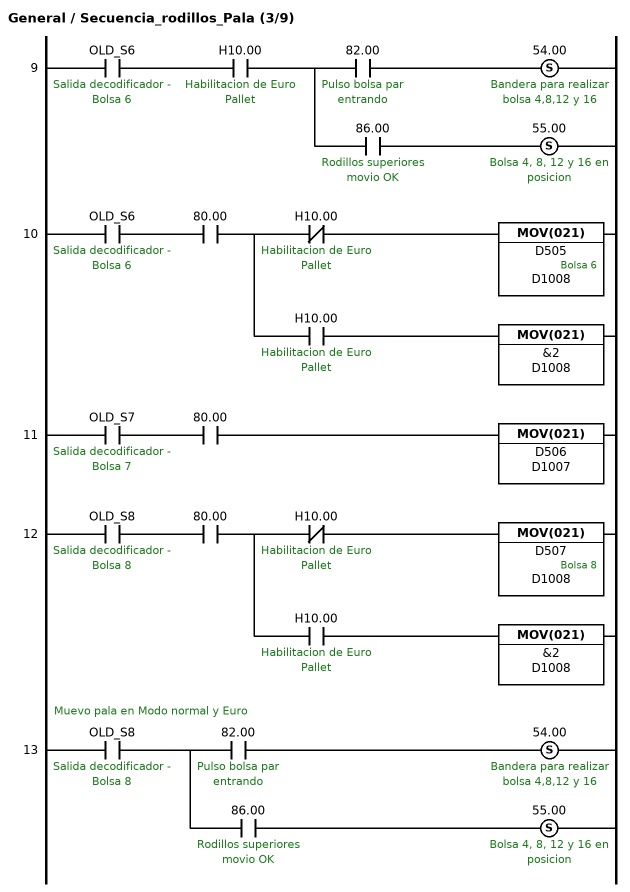
; [picture p48: General / Secuencia_rodillos_Pala, rungs 9-13]
; rung 9
LD OLD_S6  ; Salida decodificador - Bolsa 6
AND H10.00  ; Habilitacion de Euro Pallet
OUT TR0
AND 82.00  ; Pulso bolsa par entrando
SET 54.00  ; Bandera para realizar bolsa 4,8,12 y 16
LD TR0
AND 86.00  ; Rodillos superiores movio OK
SET 55.00  ; Bolsa 4, 8, 12 y 16 en posicion
; rung 10
LD OLD_S6  ; Salida decodificador - Bolsa 6
AND 80.00
OUT TR0
ANDNOT H10.00  ; Habilitacion de Euro Pallet
MOV(021) D505 D1008  ; Bolsa 6
LD TR0
AND H10.00  ; Habilitacion de Euro Pallet
MOV(021) &2 D1008
; rung 11
LD OLD_S7  ; Salida decodificador - Bolsa 7
AND 80.00
MOV(021) D506 D1007
; rung 12
LD OLD_S8  ; Salida decodificador - Bolsa 8
AND 80.00
OUT TR0
ANDNOT H10.00  ; Habilitacion de Euro Pallet
MOV(021) D507 D1008  ; Bolsa 8  // Original valor &8
LD TR0
AND H10.00  ; Habilitacion de Euro Pallet
MOV(021) &2 D1008  // Original valor &8
; rung 13: Muevo pala en Modo normal y Euro
LD OLD_S8  ; Salida decodificador - Bolsa 8
OUT TR0
AND 82.00  ; Pulso bolsa par entrando
SET 54.00  ; Bandera para realizar bolsa 4,8,12 y 16
LD TR0
AND 86.00  ; Rodillos superiores movio OK
SET 55.00  ; Bolsa 4, 8, 12 y 16 en posicion

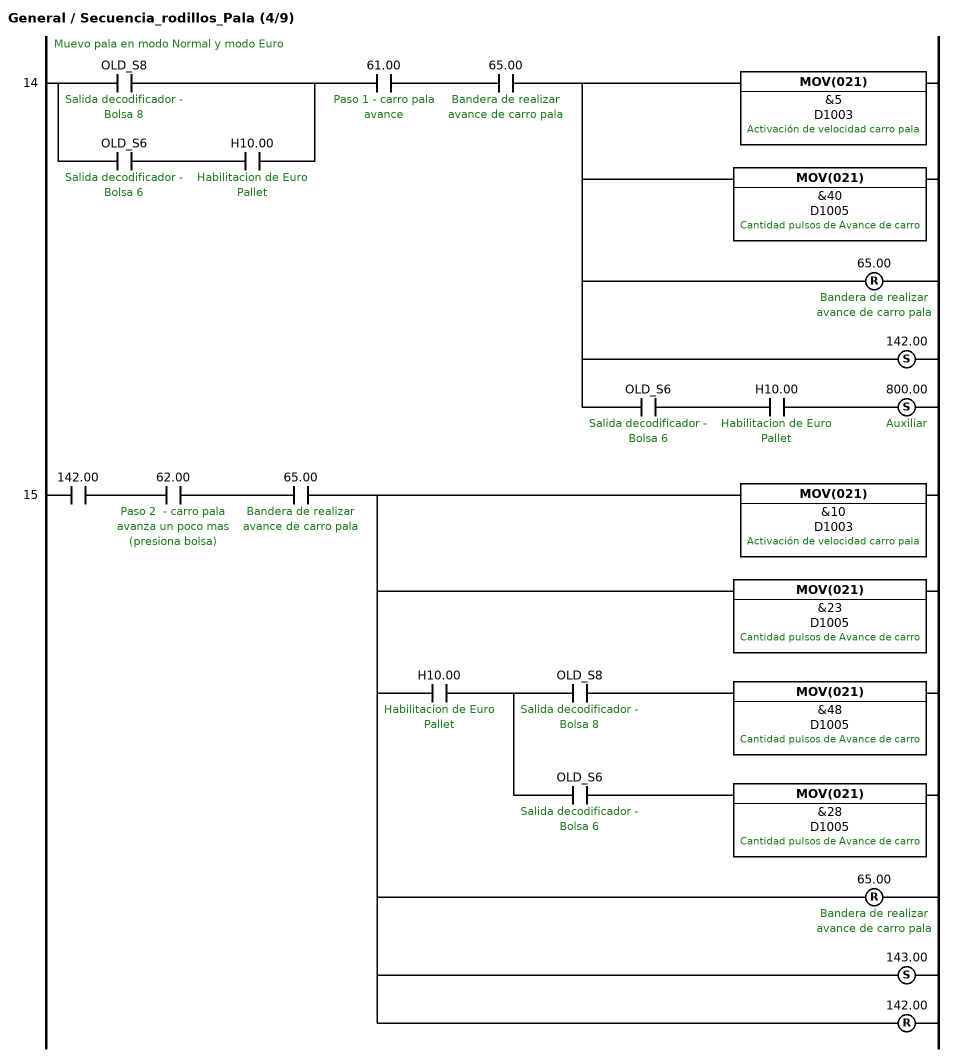
; rung 14: Muevo pala en modo Normal y modo Euro
LD OLD_S8  ; Salida decodificador - Bolsa 8
LD OLD_S6  ; Salida decodificador - Bolsa 6
AND H10.00  ; Habilitacion de Euro Pallet
ORLD
AND 61.00  ; Paso 1 - carro pala avance
AND 65.00  ; Bandera de realizar avance de carro pala
MOV(021) &5 D1003  ; Activación de velocidad carro pala
MOV(021) &40 D1005  ; Cantidad pulsos de Avance de carro
RSET 65.00  ; Bandera de realizar avance de carro pala
SET 142.00
AND OLD_S6  ; Salida decodificador - Bolsa 6
AND H10.00  ; Habilitacion de Euro Pallet
SET 800.00  ; Auxiliar
; rung 15
LD 142.00
AND 62.00  ; Paso 2  - carro pala avanza un poco mas (presiona bolsa)
AND 65.00  ; Bandera de realizar avance de carro pala
OUT TR0
MOV(021) &10 D1003  ; Activación de velocidad carro pala
MOV(021) &23 D1005  ; Cantidad pulsos de Avance de carro
AND H10.00  ; Habilitacion de Euro Pallet
OUT TR1
AND OLD_S8  ; Salida decodificador - Bolsa 8
MOV(021) &48 D1005  ; Cantidad pulsos de Avance de carro
LD TR1
AND OLD_S6  ; Salida decodificador - Bolsa 6
MOV(021) &28 D1005  ; Cantidad pulsos de Avance de carro
LD TR0
RSET 65.00  ; Bandera de realizar avance de carro pala
SET 143.00
RSET 142.00

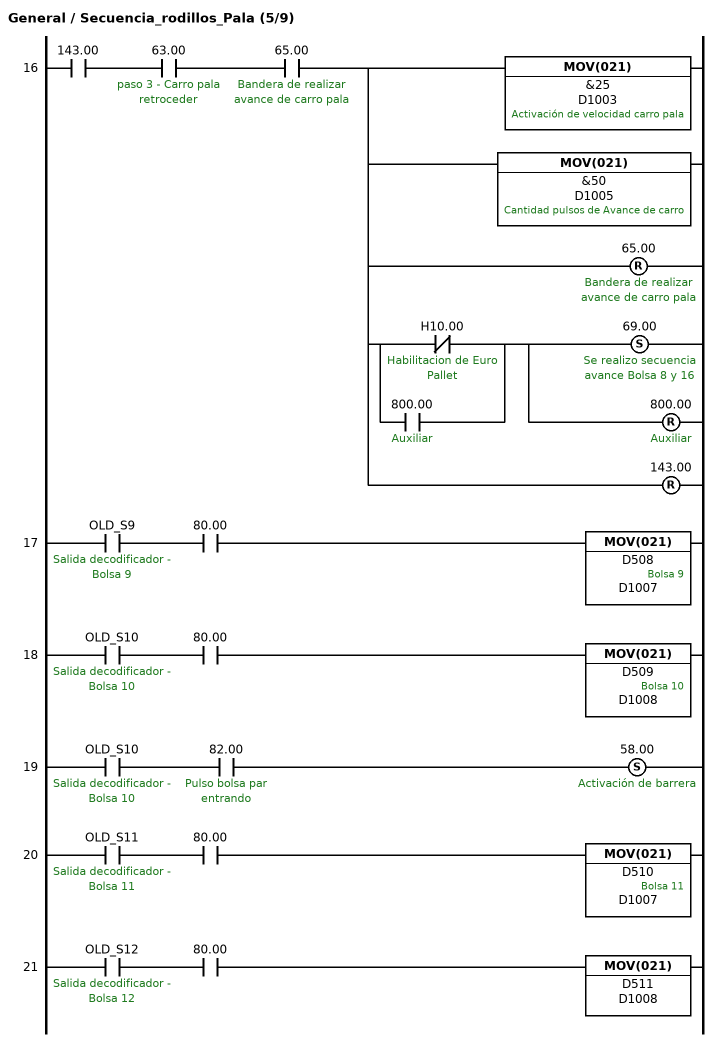
; rung 16
LD 143.00
AND 63.00  ; paso 3 - Carro pala retroceder
AND 65.00  ; Bandera de realizar avance de carro pala
OUT TR0
MOV(021) &25 D1003  ; Activación de velocidad carro pala
MOV(021) &50 D1005  ; Cantidad pulsos de Avance de carro
RSET 65.00  ; Bandera de realizar avance de carro pala
LDNOT H10.00  ; Habilitacion de Euro Pallet
OR 800.00  ; Auxiliar
ANDLD
SET 69.00  ; Se realizo secuencia avance Bolsa 8 y 16
RSET 800.00  ; Auxiliar
LD TR0
RSET 143.00
; rung 17
LD OLD_S9  ; Salida decodificador - Bolsa 9
AND 80.00
MOV(021) D508 D1007  ; Bolsa 9
; rung 18
LD OLD_S10  ; Salida decodificador - Bolsa 10
AND 80.00
MOV(021) D509 D1008  ; Bolsa 10
; rung 19
LD OLD_S10  ; Salida decodificador - Bolsa 10
AND 82.00  ; Pulso bolsa par entrando
SET 58.00  ; Activación de barrera
; rung 20
LD OLD_S11  ; Salida decodificador - Bolsa 11
AND 80.00
MOV(021) D510 D1007  ; Bolsa 11
; rung 21
LD OLD_S12  ; Salida decodificador - Bolsa 12
AND 80.00
MOV(021) D511 D1008

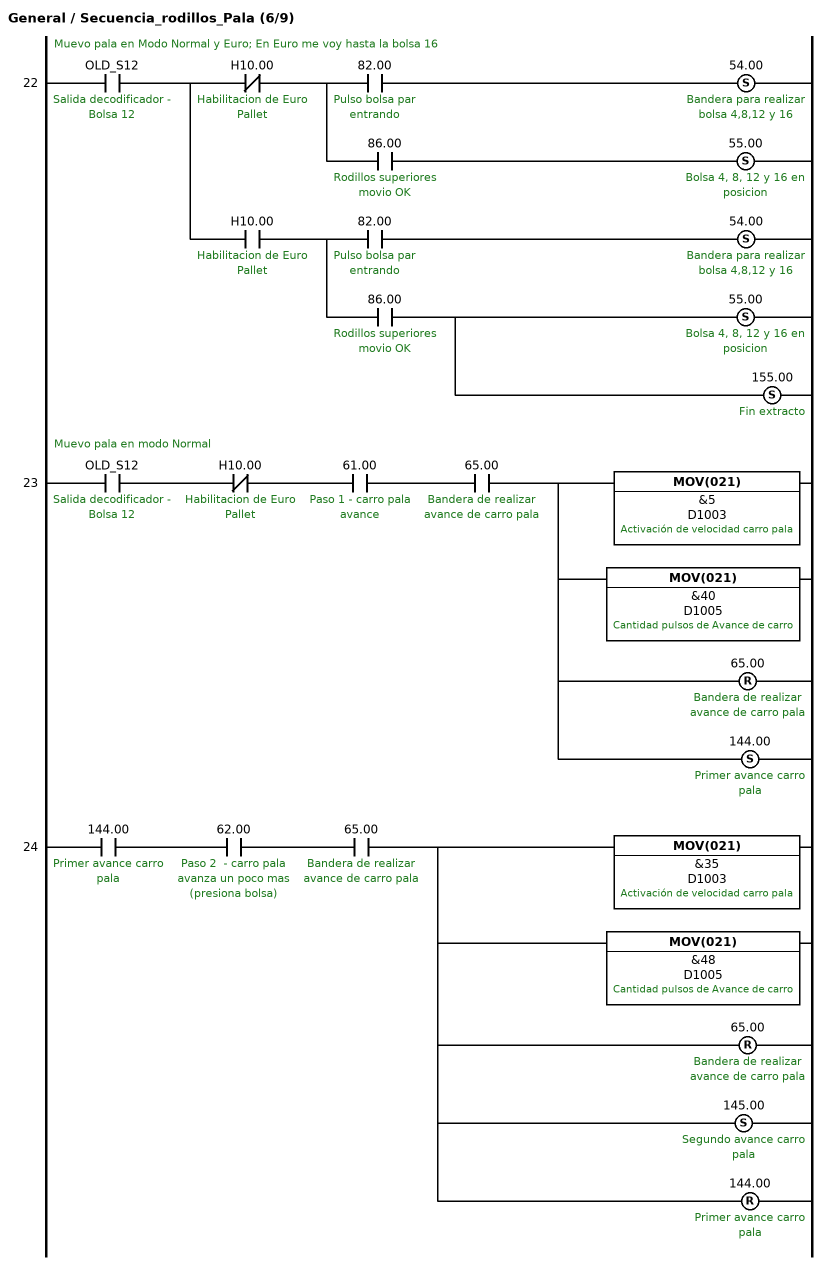
; rung 22: Muevo pala en Modo Normal y Euro; En Euro me voy hasta la bolsa 16
LD OLD_S12  ; Salida decodificador - Bolsa 12
OUT TR0
ANDNOT H10.00  ; Habilitacion de Euro Pallet
OUT TR1
AND 82.00  ; Pulso bolsa par entrando
SET 54.00  ; Bandera para realizar bolsa 4,8,12 y 16
LD TR1
AND 86.00  ; Rodillos superiores movio OK
SET 55.00  ; Bolsa 4, 8, 12 y 16 en posicion
LD TR0
AND H10.00  ; Habilitacion de Euro Pallet
OUT TR0
AND 82.00  ; Pulso bolsa par entrando
SET 54.00  ; Bandera para realizar bolsa 4,8,12 y 16
LD TR0
AND 86.00  ; Rodillos superiores movio OK
SET 55.00  ; Bolsa 4, 8, 12 y 16 en posicion
SET 155.00  ; Fin extracto
; rung 23: Muevo pala en modo Normal
LD OLD_S12  ; Salida decodificador - Bolsa 12
ANDNOT H10.00  ; Habilitacion de Euro Pallet
AND 61.00  ; Paso 1 - carro pala avance
AND 65.00  ; Bandera de realizar avance de carro pala
MOV(021) &5 D1003  ; Activación de velocidad carro pala
MOV(021) &40 D1005  ; Cantidad pulsos de Avance de carro
RSET 65.00  ; Bandera de realizar avance de carro pala
SET 144.00  ; Primer avance carro pala
; rung 24
LD 144.00  ; Primer avance carro pala
AND 62.00  ; Paso 2  - carro pala avanza un poco mas (presiona bolsa)
AND 65.00  ; Bandera de realizar avance de carro pala
MOV(021) &35 D1003  ; Activación de velocidad carro pala
MOV(021) &48 D1005  ; Cantidad pulsos de Avance de carro
RSET 65.00  ; Bandera de realizar avance de carro pala
SET 145.00  ; Segundo avance carro pala
RSET 144.00  ; Primer avance carro pala

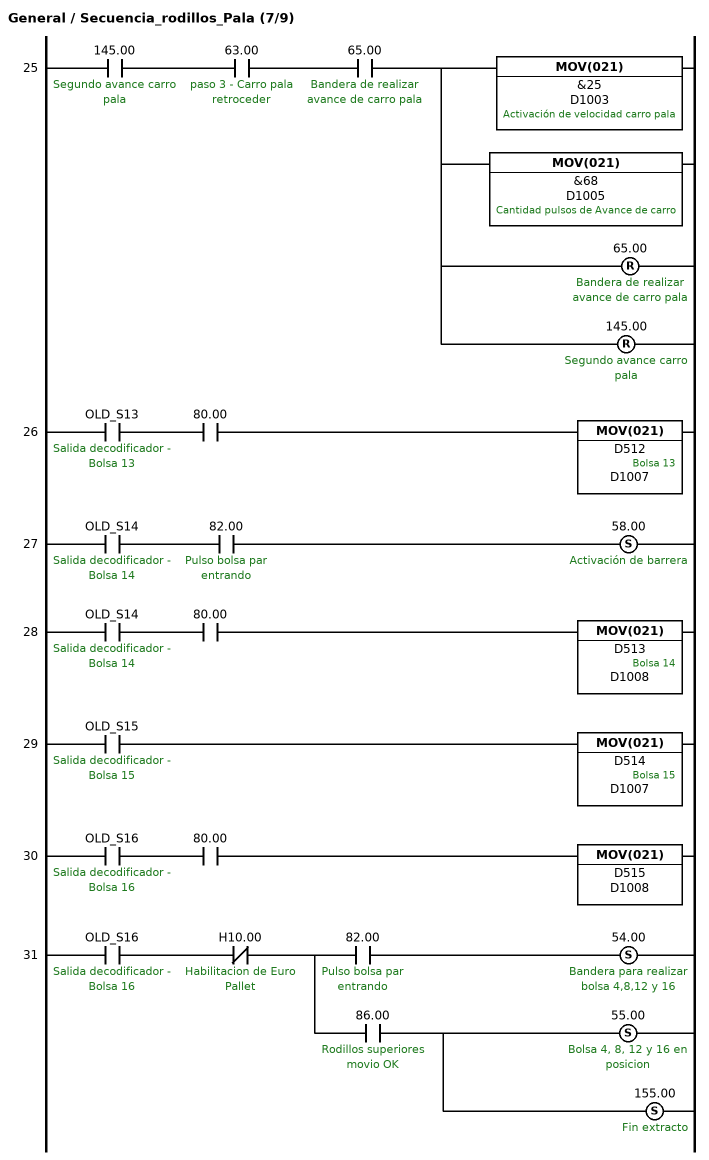
; rung 25
LD 145.00  ; Segundo avance carro pala
AND 63.00  ; paso 3 - Carro pala retroceder
AND 65.00  ; Bandera de realizar avance de carro pala
MOV(021) &25 D1003  ; Activación de velocidad carro pala
MOV(021) &68 D1005  ; Cantidad pulsos de Avance de carro
RSET 65.00  ; Bandera de realizar avance de carro pala
RSET 145.00  ; Segundo avance carro pala
; rung 26
LD OLD_S13  ; Salida decodificador - Bolsa 13
AND 80.00
MOV(021) D512 D1007  ; Bolsa 13
; rung 27
LD OLD_S14  ; Salida decodificador - Bolsa 14
AND 82.00  ; Pulso bolsa par entrando
SET 58.00  ; Activación de barrera
; rung 28
LD OLD_S14  ; Salida decodificador - Bolsa 14
AND 80.00
MOV(021) D513 D1008  ; Bolsa 14
; rung 29
LD OLD_S15  ; Salida decodificador - Bolsa 15
MOV(021) D514 D1007  ; Bolsa 15
; rung 30
LD OLD_S16  ; Salida decodificador - Bolsa 16
AND 80.00
MOV(021) D515 D1008  // Original valor &6
; rung 31
LD OLD_S16  ; Salida decodificador - Bolsa 16
ANDNOT H10.00  ; Habilitacion de Euro Pallet
OUT TR0
AND 82.00  ; Pulso bolsa par entrando
SET 54.00  ; Bandera para realizar bolsa 4,8,12 y 16
LD TR0
AND 86.00  ; Rodillos superiores movio OK
SET 55.00  ; Bolsa 4, 8, 12 y 16 en posicion
SET 155.00  ; Fin extracto

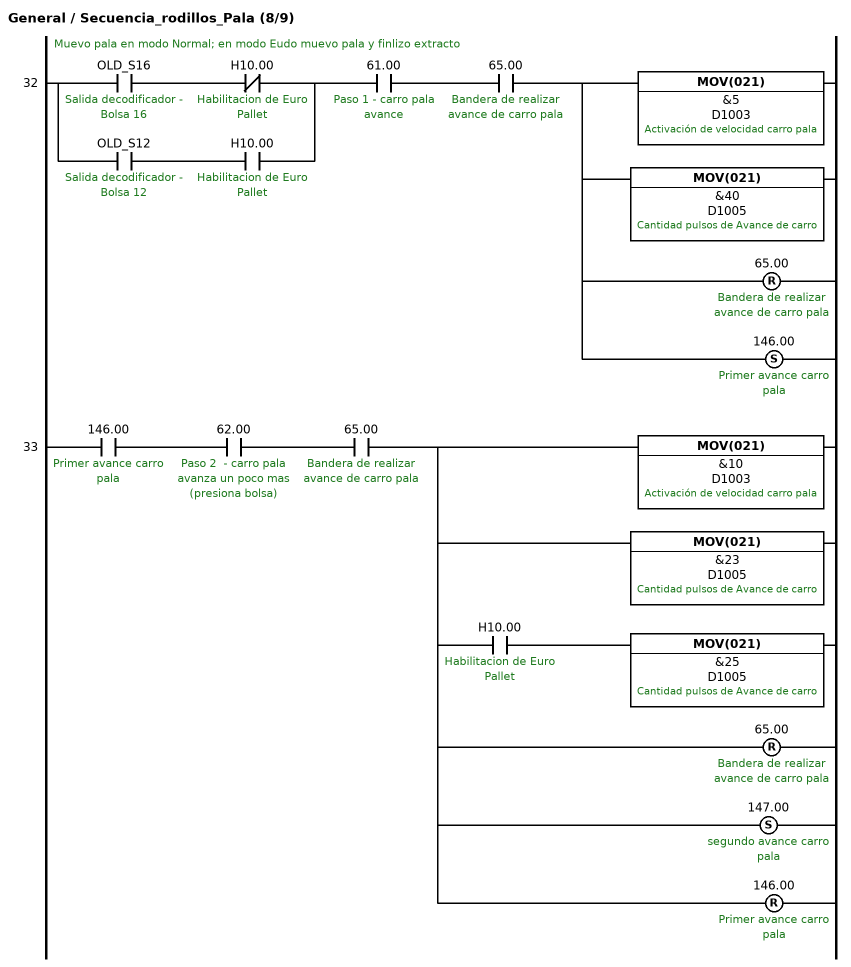
; rung 32: Muevo pala en modo Normal; en modo Eudo muevo pala y finlizo extracto
LD OLD_S16  ; Salida decodificador - Bolsa 16
ANDNOT H10.00  ; Habilitacion de Euro Pallet
LD OLD_S12  ; Salida decodificador - Bolsa 12
AND H10.00  ; Habilitacion de Euro Pallet
ORLD
AND 61.00  ; Paso 1 - carro pala avance
AND 65.00  ; Bandera de realizar avance de carro pala
MOV(021) &5 D1003  ; Activación de velocidad carro pala
MOV(021) &40 D1005  ; Cantidad pulsos de Avance de carro
RSET 65.00  ; Bandera de realizar avance de carro pala
SET 146.00  ; Primer avance carro pala
; rung 33
LD 146.00  ; Primer avance carro pala
AND 62.00  ; Paso 2  - carro pala avanza un poco mas (presiona bolsa)
AND 65.00  ; Bandera de realizar avance de carro pala
OUT TR0
MOV(021) &10 D1003  ; Activación de velocidad carro pala
MOV(021) &23 D1005  ; Cantidad pulsos de Avance de carro
AND H10.00  ; Habilitacion de Euro Pallet
MOV(021) &25 D1005  ; Cantidad pulsos de Avance de carro
LD TR0
RSET 65.00  ; Bandera de realizar avance de carro pala
SET 147.00  ; segundo avance carro pala
RSET 146.00  ; Primer avance carro pala

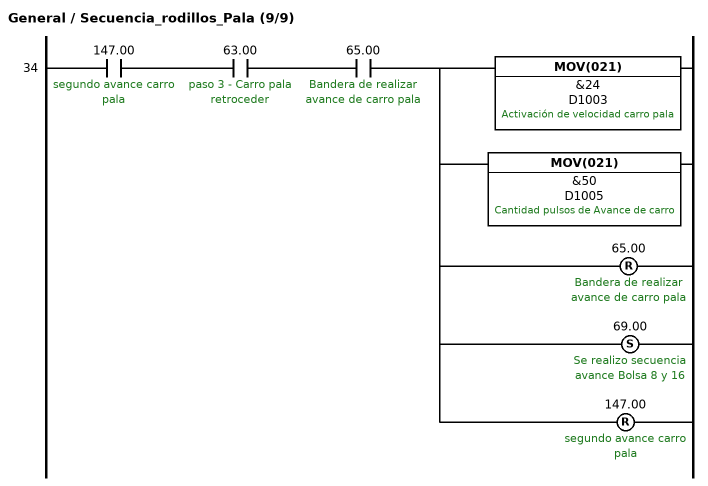
; rung 34
LD 147.00  ; segundo avance carro pala
AND 63.00  ; paso 3 - Carro pala retroceder
AND 65.00  ; Bandera de realizar avance de carro pala
MOV(021) &24 D1003  ; Activación de velocidad carro pala
MOV(021) &50 D1005  ; Cantidad pulsos de Avance de carro
RSET 65.00  ; Bandera de realizar avance de carro pala
SET 69.00  ; Se realizo secuencia avance Bolsa 8 y 16
RSET 147.00  ; segundo avance carro pala

### Section _Fin_Salto

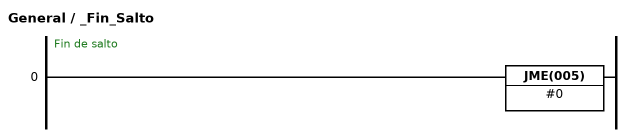
; rung 0: Fin de salto
JME(005) #0

### Section Habilitaciones_MAN_AUT

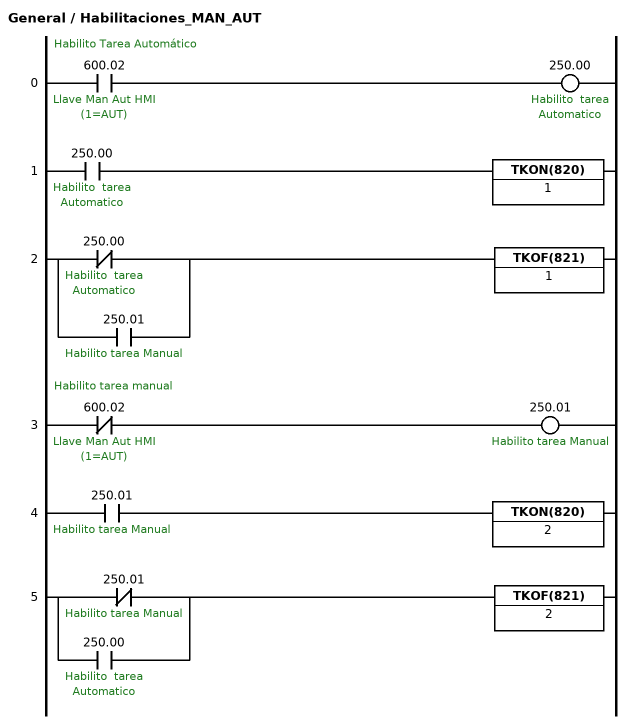
; rung 0: Habilito Tarea Automático
LD 600.02  ; Llave Man Aut HMI (1=AUT)
OUT 250.00  ; Habilito  tarea Automatico
; rung 1
LD 250.00  ; Habilito  tarea Automatico
TKON(820) 1
; rung 2
LDNOT 250.00  ; Habilito  tarea Automatico
OR 250.01  ; Habilito tarea Manual
TKOF(821) 1
; rung 3: Habilito tarea manual
LDNOT 600.02  ; Llave Man Aut HMI (1=AUT)
OUT 250.01  ; Habilito tarea Manual
; rung 4
LD 250.01  ; Habilito tarea Manual
TKON(820) 2
; rung 5
LDNOT 250.01  ; Habilito tarea Manual
OR 250.00  ; Habilito  tarea Automatico
TKOF(821) 2

### Section Seleccion_pallet

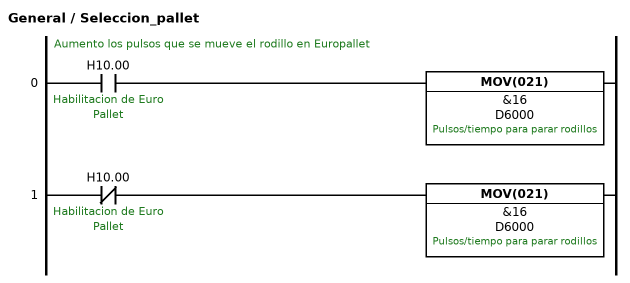
; rung 0: Aumento los pulsos que se mueve el rodillo en Europallet
LD H10.00  ; Habilitacion de Euro Pallet
MOV(021) &16 D6000  ; Pulsos/tiempo para parar rodillos
; rung 1
LDNOT H10.00  ; Habilitacion de Euro Pallet
MOV(021) &16 D6000  ; Pulsos/tiempo para parar rodillos

### Section Señales_enfundora

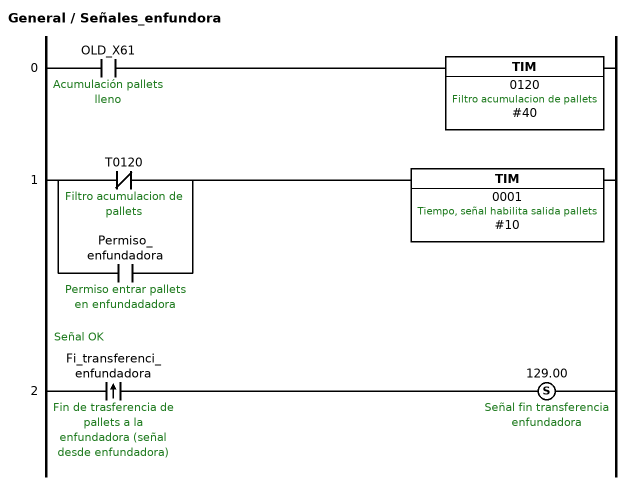
; rung 0
LD OLD_X61  ; Acumulación pallets lleno
TIM 0120 #40  ; Filtro acumulacion de pallets
; rung 1
LDNOT T0120  ; Filtro acumulacion de pallets
OR Permiso_enfundadora  ; Permiso entrar pallets en enfundadadora
TIM 0001 #10  ; Tiempo, señal habilita salida pallets
; rung 2: Señal OK
@LD Fi_transferenci_enfundadora  ; Fin de trasferencia de pallets a la enfundadora (señal desde enfundadora)
SET 129.00  ; Señal fin transferencia enfundadora

### Section Alarmas

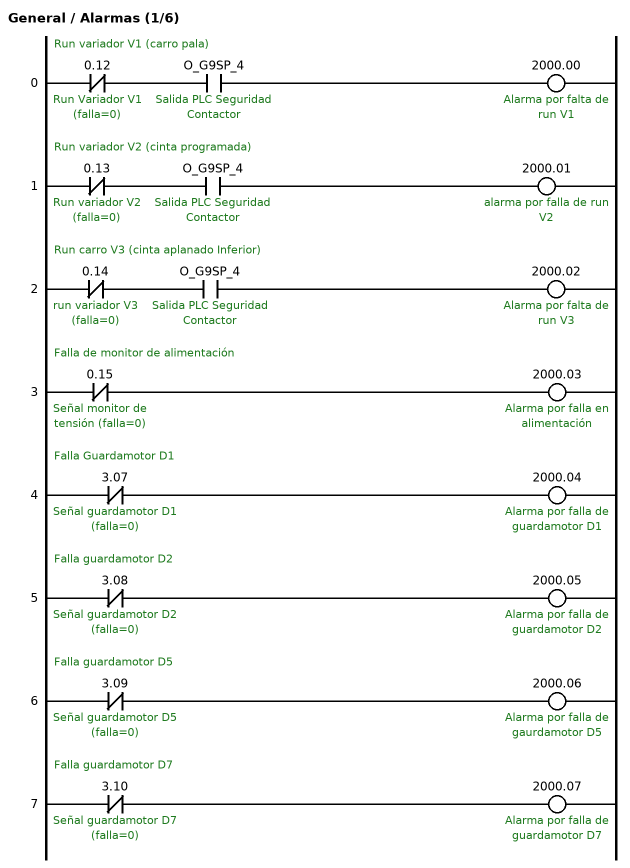
; rung 0: Run variador V1 (carro pala)
LDNOT 0.12  ; Run Variador V1 (falla=0)
AND O_G9SP_4  ; Salida PLC Seguridad Contactor
OUT 2000.00  ; Alarma por falta de run V1
; rung 1: Run variador V2 (cinta programada)
LDNOT 0.13  ; Run variador V2 (falla=0)
AND O_G9SP_4  ; Salida PLC Seguridad Contactor
OUT 2000.01  ; alarma por falla de run V2
; rung 2: Run carro V3 (cinta aplanado Inferior)
LDNOT 0.14  ; run variador V3 (falla=0)
AND O_G9SP_4  ; Salida PLC Seguridad Contactor
OUT 2000.02  ; Alarma por falta de run V3
; rung 3: Falla de monitor de alimentación
LDNOT 0.15  ; Señal monitor de tensión (falla=0)
OUT 2000.03  ; Alarma por falla en alimentación
; rung 4: Falla Guardamotor D1
LDNOT 3.07  ; Señal guardamotor D1 (falla=0)
OUT 2000.04  ; Alarma por falla de guardamotor D1
; rung 5: Falla guardamotor D2
LDNOT 3.08  ; Señal guardamotor D2 (falla=0)
OUT 2000.05  ; Alarma por falla de guardamotor D2
; rung 6: Falla guardamotor D5
LDNOT 3.09  ; Señal guardamotor D5 (falla=0)
OUT 2000.06  ; Alarma por falla de gaurdamotor D5
; rung 7: Falla guardamotor D7
LDNOT 3.10  ; Señal guardamotor D7 (falla=0)
OUT 2000.07  ; Alarma por falla de guardamotor D7

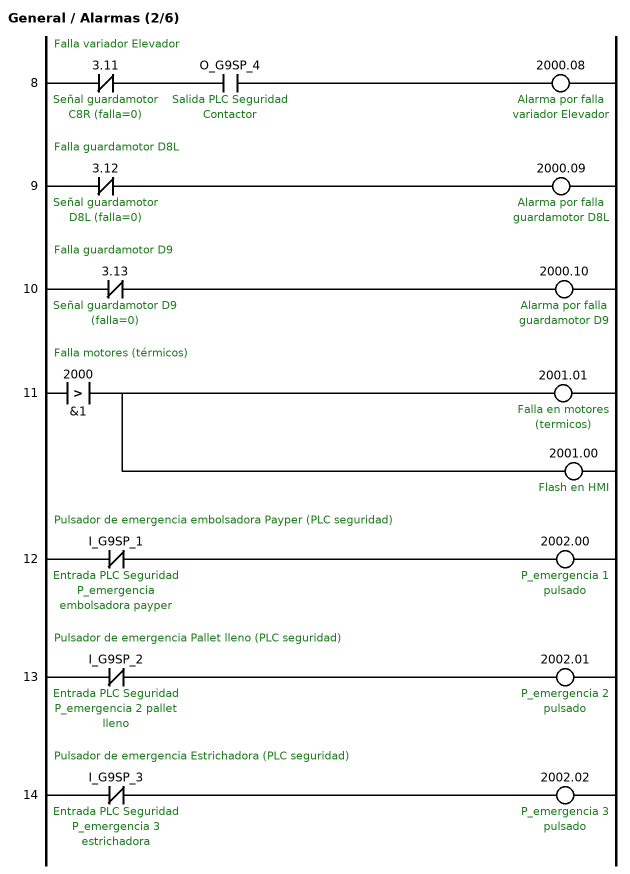
; rung 8: Falla variador Elevador
LDNOT 3.11  ; Señal guardamotor C8R (falla=0)
AND O_G9SP_4  ; Salida PLC Seguridad Contactor
OUT 2000.08  ; Alarma por falla variador Elevador
; rung 9: Falla guardamotor D8L
LDNOT 3.12  ; Señal guardamotor D8L (falla=0)
OUT 2000.09  ; Alarma por falla guardamotor D8L
; rung 10: Falla guardamotor D9
LDNOT 3.13  ; Señal guardamotor D9 (falla=0)
OUT 2000.10  ; Alarma por falla guardamotor D9
; rung 11: Falla motores (térmicos)
LD>(320) 2000 &1
OUT 2001.01  ; Falla en motores (termicos)
OUT 2001.00  ; Flash en HMI
; rung 12: Pulsador de emergencia embolsadora Payper (PLC seguridad)
LDNOT I_G9SP_1  ; Entrada PLC Seguridad P_emergencia embolsadora payper
OUT 2002.00  ; P_emergencia 1 pulsado
; rung 13: Pulsador de emergencia Pallet lleno (PLC seguridad)
LDNOT I_G9SP_2  ; Entrada PLC Seguridad P_emergencia 2 pallet lleno
OUT 2002.01  ; P_emergencia 2 pulsado
; rung 14: Pulsador de emergencia Estrichadora (PLC seguridad)
LDNOT I_G9SP_3  ; Entrada PLC Seguridad P_emergencia 3 estrichadora
OUT 2002.02  ; P_emergencia 3 pulsado

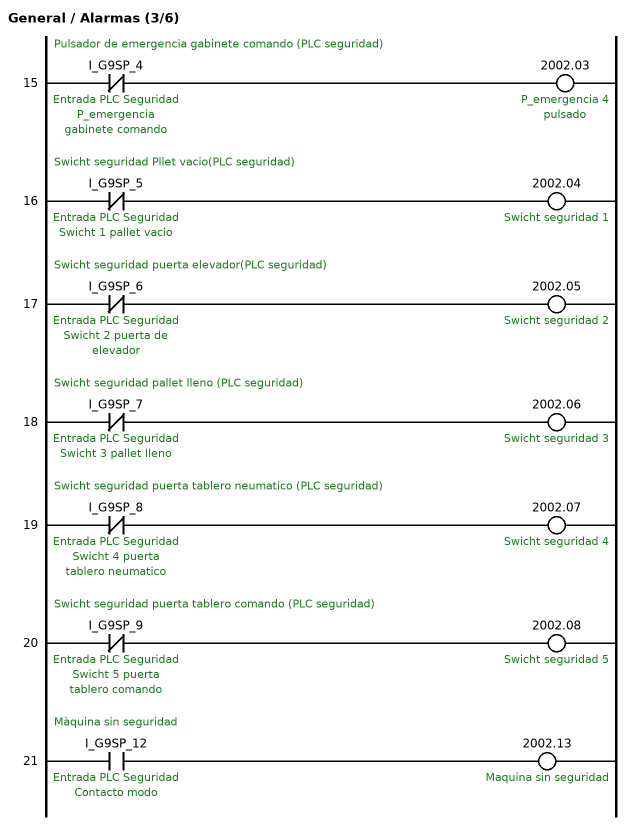
; rung 15: Pulsador de emergencia gabinete comando (PLC seguridad)
LDNOT I_G9SP_4  ; Entrada PLC Seguridad P_emergencia gabinete comando
OUT 2002.03  ; P_emergencia 4 pulsado
; rung 16: Swicht seguridad Pllet vacio(PLC seguridad)
LDNOT I_G9SP_5  ; Entrada PLC Seguridad Swicht 1 pallet vacio
OUT 2002.04  ; Swicht seguridad 1
; rung 17: Swicht seguridad puerta elevador(PLC seguridad)
LDNOT I_G9SP_6  ; Entrada PLC Seguridad Swicht 2 puerta de elevador
OUT 2002.05  ; Swicht seguridad 2
; rung 18: Swicht seguridad pallet lleno (PLC seguridad)
LDNOT I_G9SP_7  ; Entrada PLC Seguridad Swicht 3 pallet lleno
OUT 2002.06  ; Swicht seguridad 3
; rung 19: Swicht seguridad puerta tablero neumatico (PLC seguridad)
LDNOT I_G9SP_8  ; Entrada PLC Seguridad Swicht 4 puerta tablero neumatico
OUT 2002.07  ; Swicht seguridad 4
; rung 20: Swicht seguridad puerta tablero comando (PLC seguridad)
LDNOT I_G9SP_9  ; Entrada PLC Seguridad Swicht 5 puerta tablero comando
OUT 2002.08  ; Swicht seguridad 5
; rung 21: Màquina sin seguridad
LD I_G9SP_12  ; Entrada PLC Seguridad Contacto modo
OUT 2002.13  ; Maquina sin seguridad

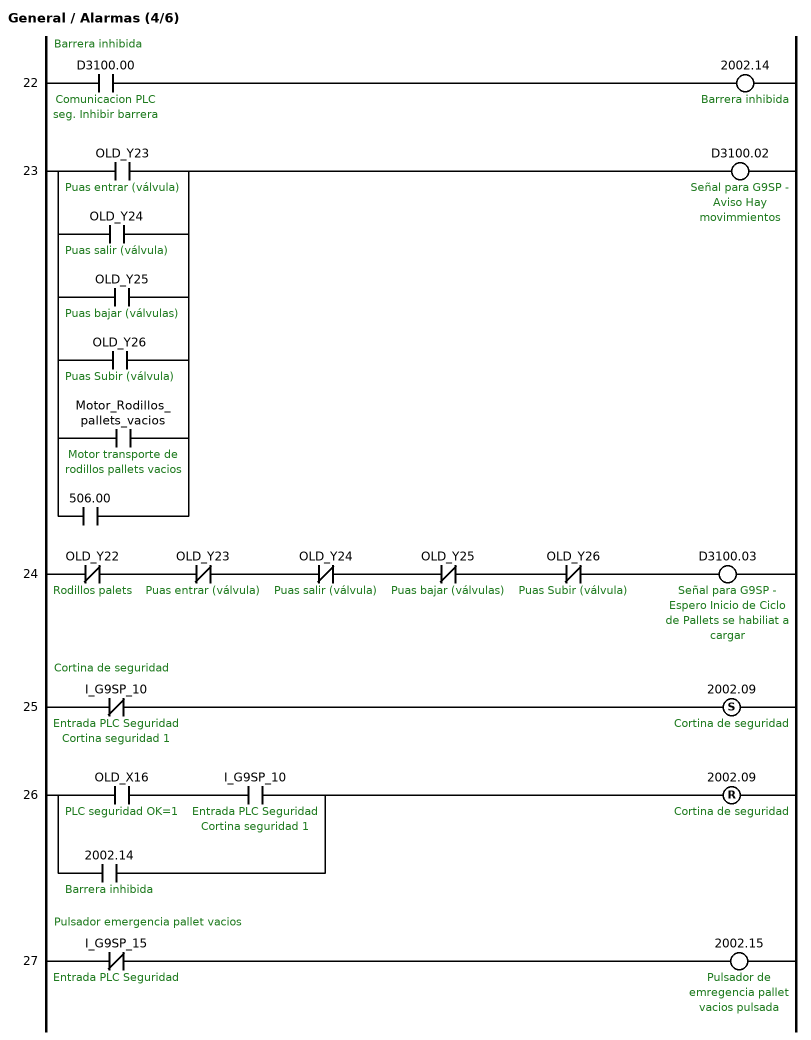
; rung 22: Barrera inhibida
LD D3100.00  ; Comunicacion PLC seg. Inhibir barrera
OUT 2002.14  ; Barrera inhibida
; rung 23
LD OLD_Y23  ; Puas entrar (válvula)
OR OLD_Y24  ; Puas salir (válvula)
OR OLD_Y25  ; Puas bajar (válvulas)
OR OLD_Y26  ; Puas Subir (válvula)
OR Motor_Rodillos_pallets_vacios  ; Motor transporte de rodillos pallets vacios
OR 506.00
OUT D3100.02  ; Señal para G9SP - Aviso Hay movimmientos
; rung 24
LDNOT OLD_Y22  ; Rodillos palets
ANDNOT OLD_Y23  ; Puas entrar (válvula)
ANDNOT OLD_Y24  ; Puas salir (válvula)
ANDNOT OLD_Y25  ; Puas bajar (válvulas)
ANDNOT OLD_Y26  ; Puas Subir (válvula)
OUT D3100.03  ; Señal para G9SP - Espero Inicio de Ciclo de Pallets se habiliat a cargar
; rung 25: Cortina de seguridad
LDNOT I_G9SP_10  ; Entrada PLC Seguridad Cortina seguridad 1
SET 2002.09  ; Cortina de seguridad
; rung 26
LD OLD_X16  ; PLC seguridad OK=1
AND I_G9SP_10  ; Entrada PLC Seguridad Cortina seguridad 1
OR 2002.14  ; Barrera inhibida
RSET 2002.09  ; Cortina de seguridad
; rung 27: Pulsador emergencia pallet vacios
LDNOT I_G9SP_15  ; Entrada PLC Seguridad
OUT 2002.15  ; Pulsador de emregencia pallet vacios pulsada

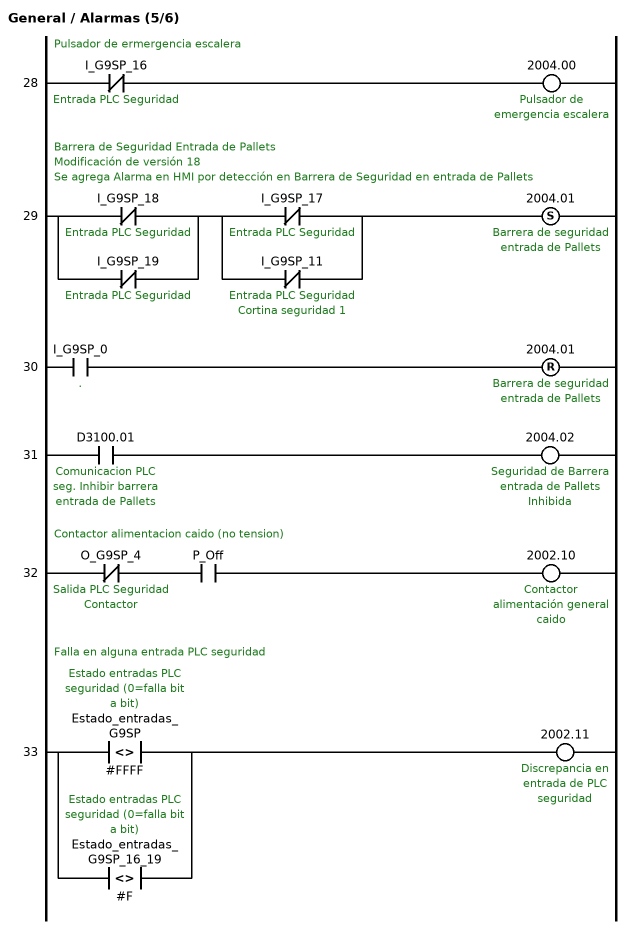
; rung 28: Pulsador de ermergencia escalera
LDNOT I_G9SP_16  ; Entrada PLC Seguridad
OUT 2004.00  ; Pulsador de emergencia escalera
; rung 29: Barrera de Seguridad Entrada de Pallets / Modificación de versión 18 / Se agrega Alarma en HMI por detección en Barrera de Seguridad en entrada de Pallets
LDNOT I_G9SP_18  ; Entrada PLC Seguridad
ORNOT I_G9SP_19  ; Entrada PLC Seguridad
LDNOT I_G9SP_17  ; Entrada PLC Seguridad
ORNOT I_G9SP_11  ; Entrada PLC Seguridad Cortina seguridad 1
ANDLD
SET 2004.01  ; Barrera de seguridad entrada de Pallets
; rung 30
LD I_G9SP_0  ; .
RSET 2004.01  ; Barrera de seguridad entrada de Pallets
; rung 31
LD D3100.01  ; Comunicacion PLC seg. Inhibir barrera entrada de Pallets
OUT 2004.02  ; Seguridad de Barrera entrada de Pallets Inhibida
; rung 32: Contactor alimentacion caido (no tension)
LDNOT O_G9SP_4  ; Salida PLC Seguridad Contactor
AND P_Off
OUT 2002.10  ; Contactor alimentación general caido
; rung 33: Falla en alguna entrada PLC seguridad
LD<>(305) Estado_entradas_G9SP #FFFF  ; Estado entradas PLC seguridad (0=falla bit a bit)
OR<>(305) Estado_entradas_G9SP_16_19 #F  ; Estado entradas PLC seguridad (0=falla bit a bit)
OUT 2002.11  ; Discrepancia en entrada de PLC seguridad

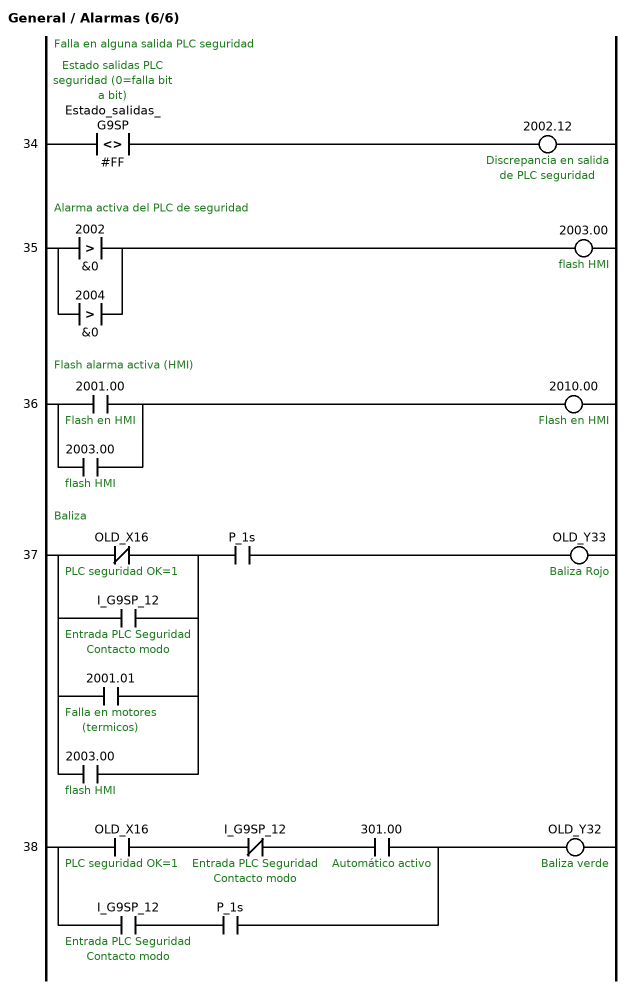
; rung 34: Falla en alguna salida PLC seguridad
LD<>(305) Estado_salidas_G9SP #FF  ; Estado salidas PLC seguridad (0=falla bit a bit)
OUT 2002.12  ; Discrepancia en salida de PLC seguridad
; rung 35: Alarma activa del PLC de seguridad
LD>(320) 2002 &0
OR>(320) 2004 &0
OUT 2003.00  ; flash HMI
; rung 36: Flash alarma activa (HMI)
LD 2001.00  ; Flash en HMI
OR 2003.00  ; flash HMI
OUT 2010.00  ; Flash en HMI
; rung 37: Baliza
LDNOT OLD_X16  ; PLC seguridad OK=1
OR I_G9SP_12  ; Entrada PLC Seguridad Contacto modo
OR 2001.01  ; Falla en motores (termicos)
OR 2003.00  ; flash HMI
AND P_1s
OUT OLD_Y33  ; Baliza Rojo
; rung 38
LD OLD_X16  ; PLC seguridad OK=1
ANDNOT I_G9SP_12  ; Entrada PLC Seguridad Contacto modo
AND 301.00  ; Automático activo
LD I_G9SP_12  ; Entrada PLC Seguridad Contacto modo
AND P_1s
ORLD
OUT OLD_Y32  ; Baliza verde

### Section Salidas_seguras

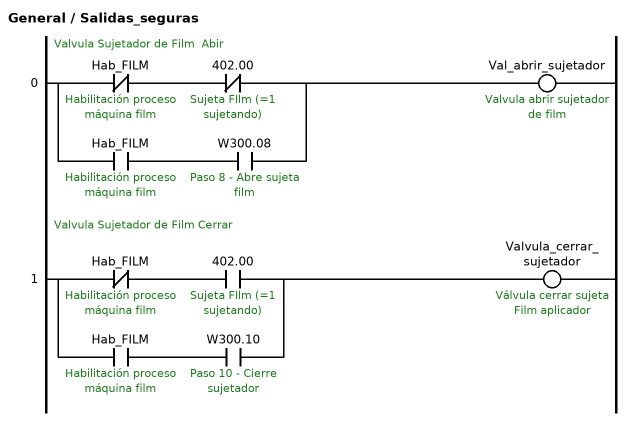
; rung 0: Valvula Sujetador de Film  Abir
LDNOT Hab_FILM  ; Habilitación proceso máquina film
ANDNOT 402.00  ; Sujeta FIlm (=1 sujetando)
LD Hab_FILM  ; Habilitación proceso máquina film
AND W300.08  ; Paso 8 - Abre sujeta film
ORLD
OUT Val_abrir_sujetador  ; Valvula abrir sujetador de film
; rung 1: Valvula Sujetador de Film Cerrar
LDNOT Hab_FILM  ; Habilitación proceso máquina film
AND 402.00  ; Sujeta FIlm (=1 sujetando)
LD Hab_FILM  ; Habilitación proceso máquina film
AND W300.10  ; Paso 10 - Cierre sujetador
ORLD
OUT Valvula_cerrar_sujetador  ; Válvula cerrar sujeta Film aplicador

### Section END
; rung 0
END(001)

## Program Automatico (cyclic task 1)

### Section Salidas_Automatico

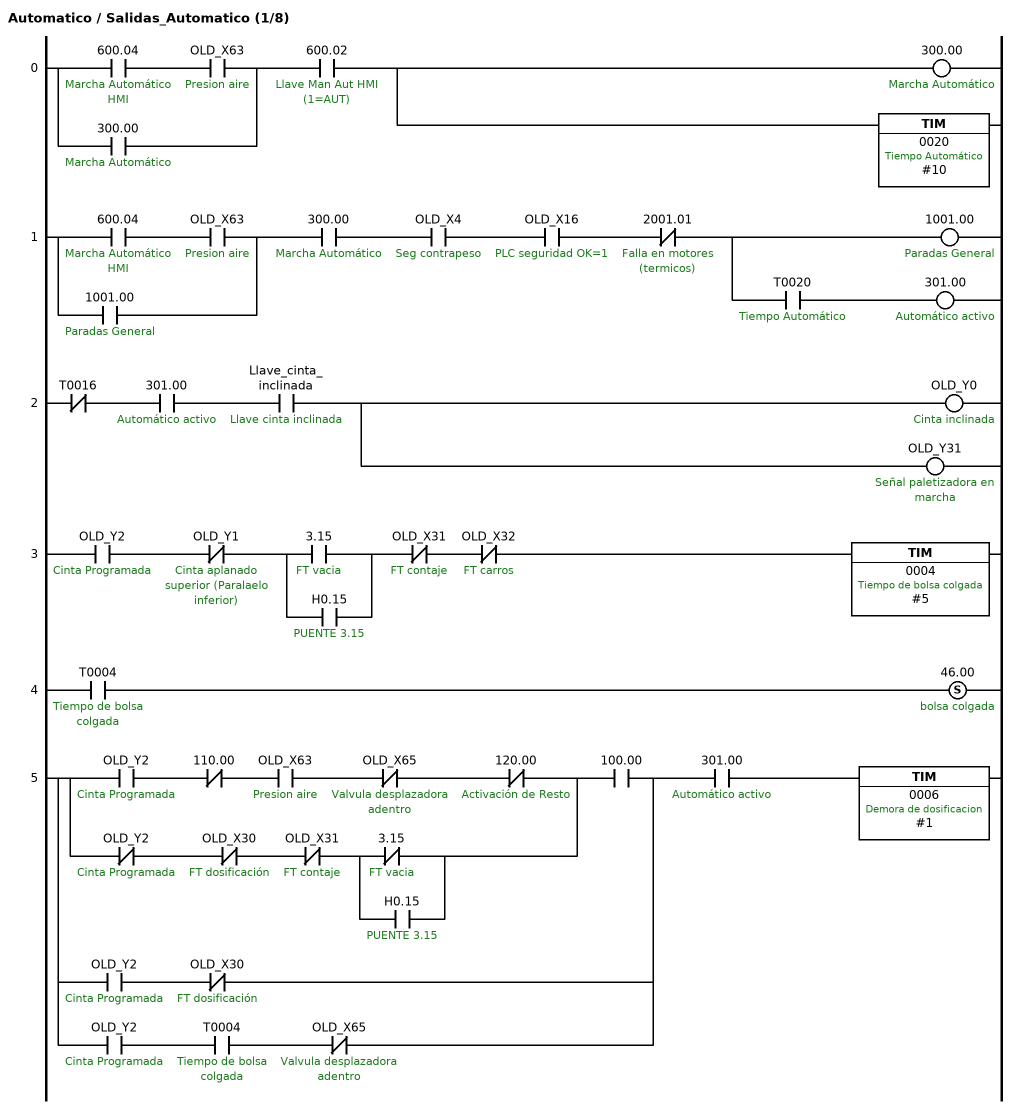
; rung 0
LD 600.04  ; Marcha Automático HMI
AND OLD_X63  ; Presion aire
OR 300.00  ; Marcha Automático
AND 600.02  ; Llave Man Aut HMI (1=AUT)
OUT 300.00  ; Marcha Automático
TIM 0020 #10  ; Tiempo Automático
; rung 1
LD 600.04  ; Marcha Automático HMI
AND OLD_X63  ; Presion aire
OR 1001.00  ; Paradas General
AND 300.00  ; Marcha Automático
AND OLD_X4  ; Seg contrapeso
AND OLD_X16  ; PLC seguridad OK=1
ANDNOT 2001.01  ; Falla en motores (termicos)
OUT 1001.00  ; Paradas General
AND T0020  ; Tiempo Automático
OUT 301.00  ; Automático activo
; rung 2
LDNOT T0016
AND 301.00  ; Automático activo
AND Llave_cinta_inclinada  ; Llave cinta inclinada
OUT OLD_Y0  ; Cinta inclinada
OUT OLD_Y31  ; Señal paletizadora en marcha
; rung 3
LD OLD_Y2  ; Cinta Programada
ANDNOT OLD_Y1  ; Cinta aplanado superior (Paralaelo inferior)
LD 3.15  ; FT vacia
OR H0.15  ; PUENTE 3.15
ANDLD
ANDNOT OLD_X31  ; FT contaje
ANDNOT OLD_X32  ; FT carros
TIM 0004 #5  ; Tiempo de bolsa colgada
; rung 4
LD T0004  ; Tiempo de bolsa colgada
SET 46.00  ; bolsa colgada
; rung 5
LD OLD_Y2  ; Cinta Programada
ANDNOT 110.00
AND OLD_X63  ; Presion aire
ANDNOT OLD_X65  ; Valvula desplazadora adentro
ANDNOT 120.00  ; Activación de Resto
LDNOT OLD_Y2  ; Cinta Programada
ANDNOT OLD_X30  ; FT dosificación
ANDNOT OLD_X31  ; FT contaje
LDNOT 3.15  ; FT vacia
OR H0.15  ; PUENTE 3.15
ANDLD
ORLD
AND 100.00
LD OLD_Y2  ; Cinta Programada
ANDNOT OLD_X30  ; FT dosificación
ORLD
LD OLD_Y2  ; Cinta Programada
AND T0004  ; Tiempo de bolsa colgada
ANDNOT OLD_X65  ; Valvula desplazadora adentro
ORLD
AND 301.00  ; Automático activo
TIM 0006 #1  ; Demora de dosificacion

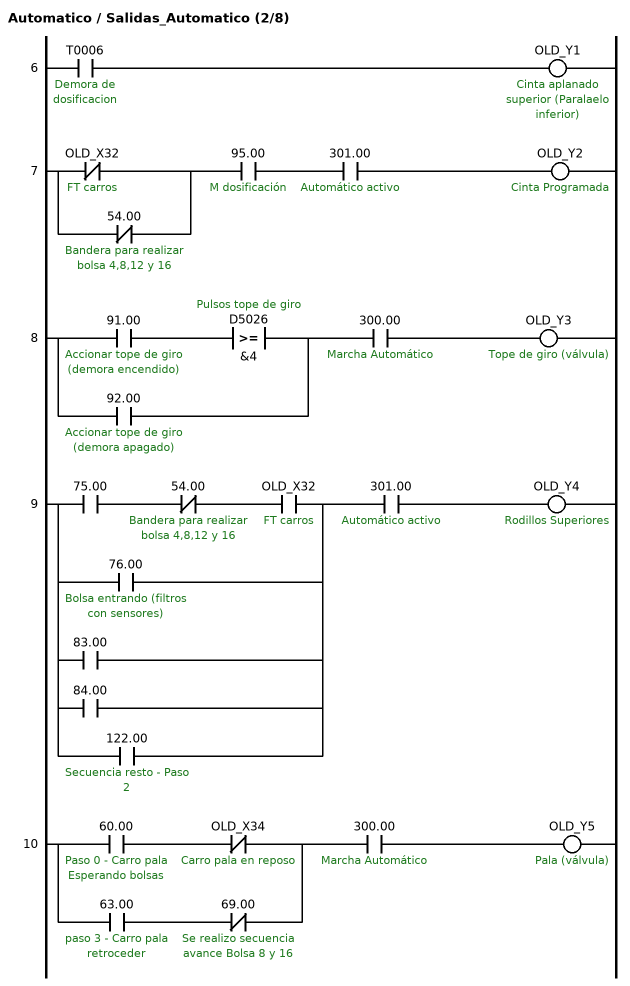
; rung 6
LD T0006  ; Demora de dosificacion
OUT OLD_Y1  ; Cinta aplanado superior (Paralaelo inferior)
; rung 7
LDNOT OLD_X32  ; FT carros
ORNOT 54.00  ; Bandera para realizar bolsa 4,8,12 y 16
AND 95.00  ; M dosificación
AND 301.00  ; Automático activo
OUT OLD_Y2  ; Cinta Programada
; rung 8
LD 91.00  ; Accionar tope de giro (demora encendido)
AND>=(325) D5026 &4  ; Pulsos tope de giro
OR 92.00  ; Accionar tope de giro (demora apagado)
AND 300.00  ; Marcha Automático
OUT OLD_Y3  ; Tope de giro (válvula)
; rung 9
LD 75.00
ANDNOT 54.00  ; Bandera para realizar bolsa 4,8,12 y 16
AND OLD_X32  ; FT carros
OR 76.00  ; Bolsa entrando (filtros con sensores)
OR 83.00
OR 84.00
OR 122.00  ; Secuencia resto - Paso 2
AND 301.00  ; Automático activo
OUT OLD_Y4  ; Rodillos Superiores
; rung 10
LD 60.00  ; Paso 0 - Carro pala Esperando bolsas
ANDNOT OLD_X34  ; Carro pala en reposo
LD 63.00  ; paso 3 - Carro pala retroceder
ANDNOT 69.00  ; Se realizo secuencia avance Bolsa 8 y 16
ORLD
AND 300.00  ; Marcha Automático
OUT OLD_Y5  ; Pala (válvula)

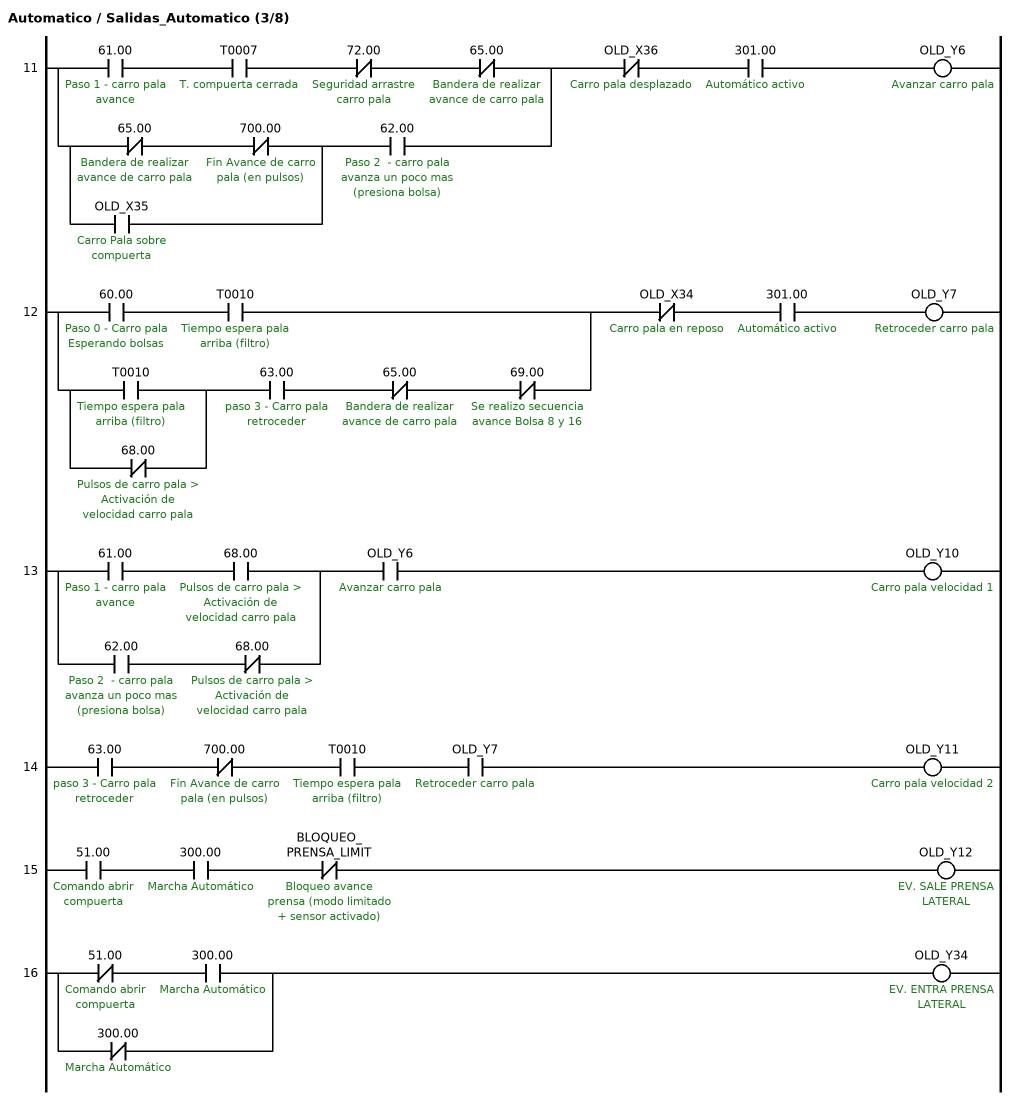
; rung 11
LD 61.00  ; Paso 1 - carro pala avance
AND T0007  ; T. compuerta cerrada
ANDNOT 72.00  ; Seguridad arrastre carro pala
ANDNOT 65.00  ; Bandera de realizar avance de carro pala
LDNOT 65.00  ; Bandera de realizar avance de carro pala
ANDNOT 700.00  ; Fin Avance de carro pala (en pulsos)
OR OLD_X35  ; Carro Pala sobre compuerta
AND 62.00  ; Paso 2  - carro pala avanza un poco mas (presiona bolsa)
ORLD
ANDNOT OLD_X36  ; Carro pala desplazado
AND 301.00  ; Automático activo
OUT OLD_Y6  ; Avanzar carro pala
; rung 12
LD 60.00  ; Paso 0 - Carro pala Esperando bolsas
AND T0010  ; Tiempo espera pala arriba (filtro)
LD T0010  ; Tiempo espera pala arriba (filtro)
ORNOT 68.00  ; Pulsos de carro pala > Activación de velocidad carro pala
AND 63.00  ; paso 3 - Carro pala retroceder
ANDNOT 65.00  ; Bandera de realizar avance de carro pala
ANDNOT 69.00  ; Se realizo secuencia avance Bolsa 8 y 16
ORLD
ANDNOT OLD_X34  ; Carro pala en reposo
AND 301.00  ; Automático activo
OUT OLD_Y7  ; Retroceder carro pala
; rung 13
LD 61.00  ; Paso 1 - carro pala avance
AND 68.00  ; Pulsos de carro pala > Activación de velocidad carro pala
LD 62.00  ; Paso 2  - carro pala avanza un poco mas (presiona bolsa)
ANDNOT 68.00  ; Pulsos de carro pala > Activación de velocidad carro pala
ORLD
AND OLD_Y6  ; Avanzar carro pala
OUT OLD_Y10  ; Carro pala velocidad 1
; rung 14
LD 63.00  ; paso 3 - Carro pala retroceder
ANDNOT 700.00  ; Fin Avance de carro pala (en pulsos)
AND T0010  ; Tiempo espera pala arriba (filtro)
AND OLD_Y7  ; Retroceder carro pala
OUT OLD_Y11  ; Carro pala velocidad 2
; rung 15
LD 51.00  ; Comando abrir compuerta
AND 300.00  ; Marcha Automático
ANDNOT BLOQUEO_PRENSA_LIMIT  ; Bloqueo avance prensa (modo limitado + sensor activado)
OUT OLD_Y12  ; EV. SALE PRENSA LATERAL
; rung 16
LDNOT 51.00  ; Comando abrir compuerta
AND 300.00  ; Marcha Automático
ORNOT 300.00  ; Marcha Automático
OUT OLD_Y34  ; EV. ENTRA PRENSA LATERAL

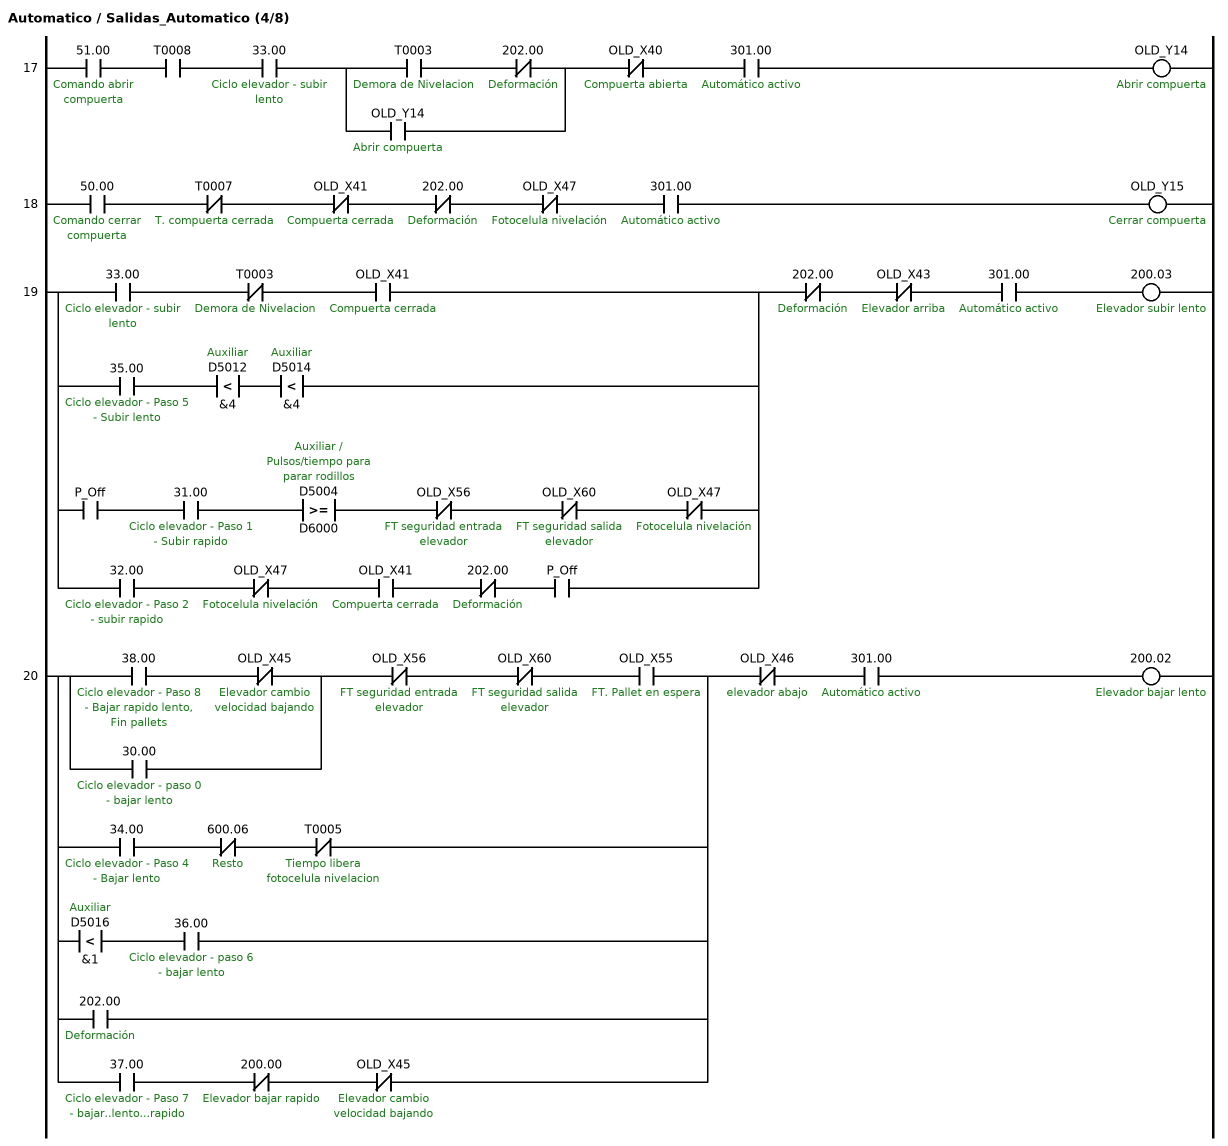
; rung 17
LD 51.00  ; Comando abrir compuerta
AND T0008
AND 33.00  ; Ciclo elevador - subir lento
LD T0003  ; Demora de Nivelacion
ANDNOT 202.00  ; Deformación
OR OLD_Y14  ; Abrir compuerta
ANDLD
ANDNOT OLD_X40  ; Compuerta abierta
AND 301.00  ; Automático activo
OUT OLD_Y14  ; Abrir compuerta
; rung 18
LD 50.00  ; Comando cerrar compuerta
ANDNOT T0007  ; T. compuerta cerrada
ANDNOT OLD_X41  ; Compuerta cerrada
ANDNOT 202.00  ; Deformación
ANDNOT OLD_X47  ; Fotocelula nivelación
AND 301.00  ; Automático activo
OUT OLD_Y15  ; Cerrar compuerta
; rung 19
LD 33.00  ; Ciclo elevador - subir lento
ANDNOT T0003  ; Demora de Nivelacion
AND OLD_X41  ; Compuerta cerrada
LD 35.00  ; Ciclo elevador - Paso 5 - Subir lento
AND<(310) D5012 &4  ; Auxiliar
AND<(310) D5014 &4  ; Auxiliar
ORLD
LD P_Off
AND 31.00  ; Ciclo elevador - Paso 1 - Subir rapido
AND>=(325) D5004 D6000  ; Auxiliar, Pulsos/tiempo para parar rodillos
ANDNOT OLD_X56  ; FT seguridad entrada elevador
ANDNOT OLD_X60  ; FT seguridad salida elevador
ANDNOT OLD_X47  ; Fotocelula nivelación
ORLD
LD 32.00  ; Ciclo elevador - Paso 2 - subir rapido
ANDNOT OLD_X47  ; Fotocelula nivelación
AND OLD_X41  ; Compuerta cerrada
ANDNOT 202.00  ; Deformación
AND P_Off
ORLD
ANDNOT 202.00  ; Deformación
ANDNOT OLD_X43  ; Elevador arriba
AND 301.00  ; Automático activo
OUT 200.03  ; Elevador subir lento
; rung 20
LD 38.00  ; Ciclo elevador - Paso 8 - Bajar rapido lento, Fin pallets
ANDNOT OLD_X45  ; Elevador cambio velocidad bajando
OR 30.00  ; Ciclo elevador - paso 0 - bajar lento
ANDNOT OLD_X56  ; FT seguridad entrada elevador
ANDNOT OLD_X60  ; FT seguridad salida elevador
AND OLD_X55  ; FT. Pallet en espera
LD 34.00  ; Ciclo elevador - Paso 4 - Bajar lento
ANDNOT 600.06  ; Resto
ANDNOT T0005  ; Tiempo libera fotocelula nivelacion
ORLD
LD<(310) D5016 &1  ; Auxiliar
AND 36.00  ; Ciclo elevador - paso 6 - bajar lento
ORLD
OR 202.00  ; Deformación
LD 37.00  ; Ciclo elevador - Paso 7 - bajar..lento...rapido
ANDNOT 200.00  ; Elevador bajar rapido
ANDNOT OLD_X45  ; Elevador cambio velocidad bajando
ORLD
ANDNOT OLD_X46  ; elevador abajo
AND 301.00  ; Automático activo
OUT 200.02  ; Elevador bajar lento

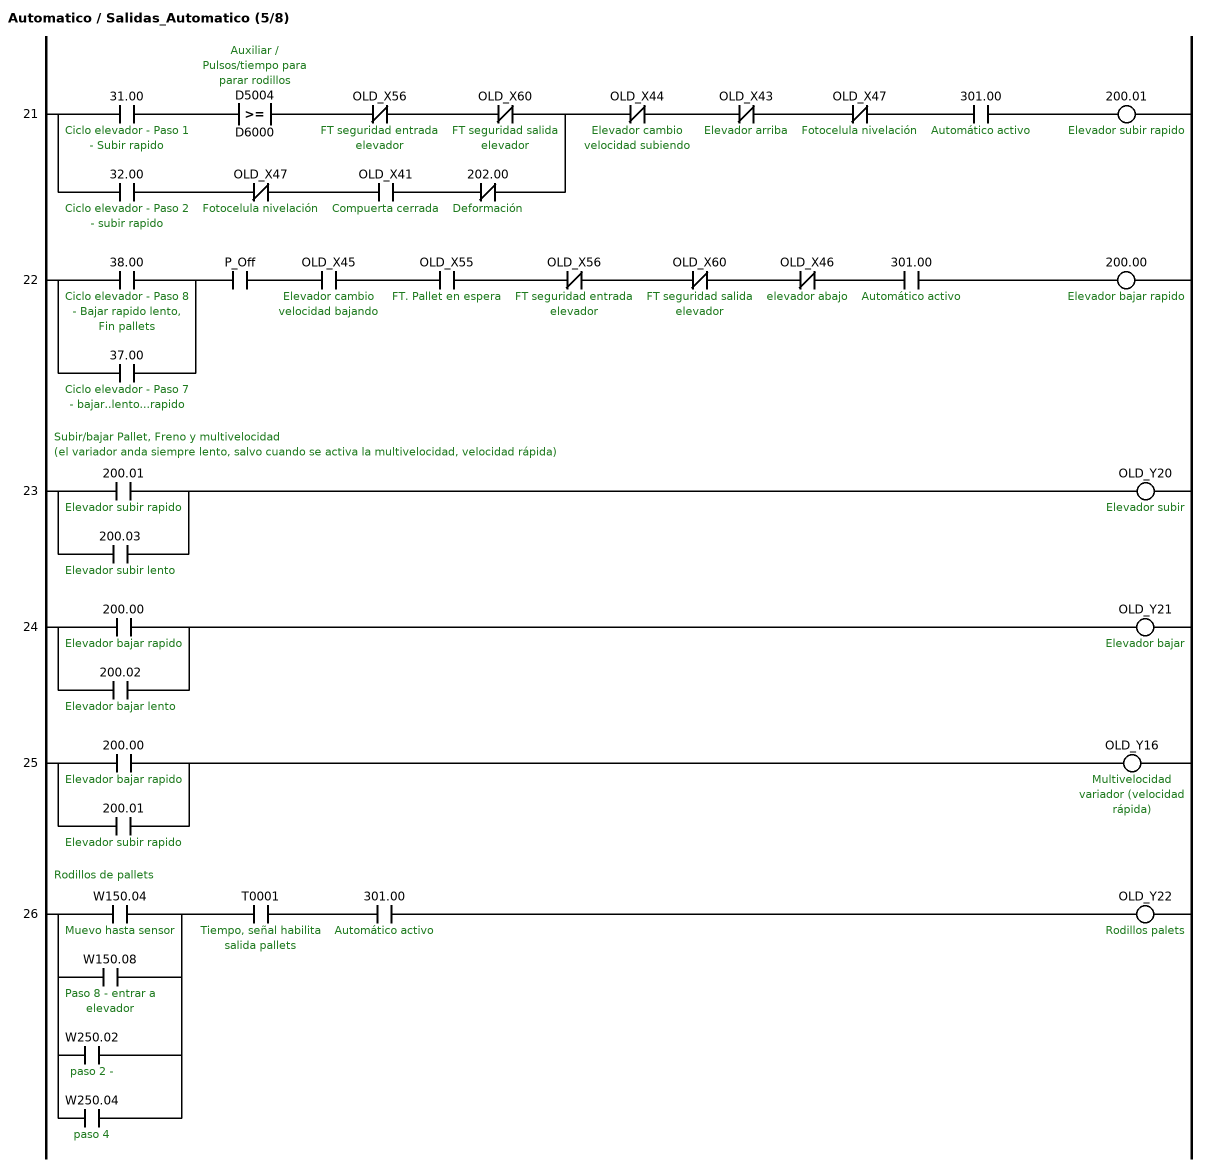
; rung 21
LD 31.00  ; Ciclo elevador - Paso 1 - Subir rapido
AND>=(325) D5004 D6000  ; Auxiliar, Pulsos/tiempo para parar rodillos
ANDNOT OLD_X56  ; FT seguridad entrada elevador
ANDNOT OLD_X60  ; FT seguridad salida elevador
LD 32.00  ; Ciclo elevador - Paso 2 - subir rapido
ANDNOT OLD_X47  ; Fotocelula nivelación
AND OLD_X41  ; Compuerta cerrada
ANDNOT 202.00  ; Deformación
ORLD
ANDNOT OLD_X44  ; Elevador cambio velocidad subiendo
ANDNOT OLD_X43  ; Elevador arriba
ANDNOT OLD_X47  ; Fotocelula nivelación
AND 301.00  ; Automático activo
OUT 200.01  ; Elevador subir rapido
; rung 22
LD 38.00  ; Ciclo elevador - Paso 8 - Bajar rapido lento, Fin pallets
OR 37.00  ; Ciclo elevador - Paso 7 - bajar..lento...rapido
AND P_Off
AND OLD_X45  ; Elevador cambio velocidad bajando
AND OLD_X55  ; FT. Pallet en espera
ANDNOT OLD_X56  ; FT seguridad entrada elevador
ANDNOT OLD_X60  ; FT seguridad salida elevador
ANDNOT OLD_X46  ; elevador abajo
AND 301.00  ; Automático activo
OUT 200.00  ; Elevador bajar rapido
; rung 23: Subir/bajar Pallet, Freno y multivelocidad / (el variador anda siempre lento, salvo cuando se activa la multivelocidad, velocidad rápida)
LD 200.01  ; Elevador subir rapido
OR 200.03  ; Elevador subir lento
OUT OLD_Y20  ; Elevador subir
; rung 24
LD 200.00  ; Elevador bajar rapido
OR 200.02  ; Elevador bajar lento
OUT OLD_Y21  ; Elevador bajar
; rung 25
LD 200.00  ; Elevador bajar rapido
OR 200.01  ; Elevador subir rapido
OUT OLD_Y16  ; Multivelocidad variador (velocidad rápida)
; rung 26: Rodillos de pallets
LD W150.04  ; Muevo hasta sensor
OR W150.08  ; Paso 8 - entrar a elevador
OR W250.02  ; paso 2 -
OR W250.04  ; paso 4
AND T0001  ; Tiempo, señal habilita salida pallets
AND 301.00  ; Automático activo
OUT OLD_Y22  ; Rodillos palets

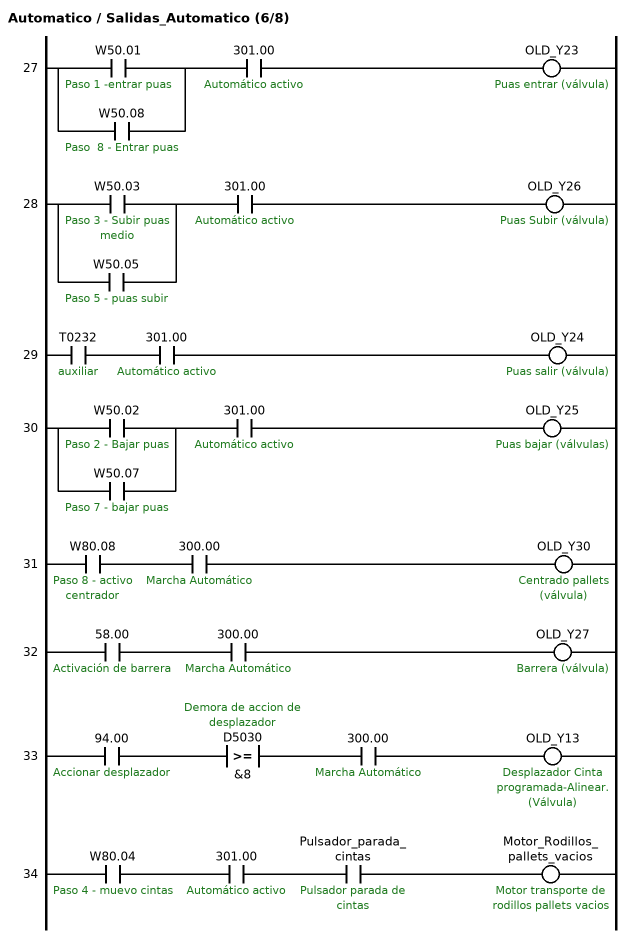
; rung 27
LD W50.01  ; Paso 1 -entrar puas
OR W50.08  ; Paso  8 - Entrar puas
AND 301.00  ; Automático activo
OUT OLD_Y23  ; Puas entrar (válvula)
; rung 28
LD W50.03  ; Paso 3 - Subir puas medio
OR W50.05  ; Paso 5 - puas subir
AND 301.00  ; Automático activo
OUT OLD_Y26  ; Puas Subir (válvula)
; rung 29
LD T0232  ; auxiliar
AND 301.00  ; Automático activo
OUT OLD_Y24  ; Puas salir (válvula)
; rung 30
LD W50.02  ; Paso 2 - Bajar puas
OR W50.07  ; Paso 7 - bajar puas
AND 301.00  ; Automático activo
OUT OLD_Y25  ; Puas bajar (válvulas)
; rung 31
LD W80.08  ; Paso 8 - activo centrador
AND 300.00  ; Marcha Automático
OUT OLD_Y30  ; Centrado pallets (válvula)
; rung 32
LD 58.00  ; Activación de barrera
AND 300.00  ; Marcha Automático
OUT OLD_Y27  ; Barrera (válvula)
; rung 33
LD 94.00  ; Accionar desplazador
AND>=(325) D5030 &8  ; Demora de accion de desplazador
AND 300.00  ; Marcha Automático
OUT OLD_Y13  ; Desplazador Cinta programada-Alinear. (Válvula)
; rung 34
LD W80.04  ; Paso 4 - muevo cintas
AND 301.00  ; Automático activo
AND Pulsador_parada_cintas  ; Pulsador parada de cintas
OUT Motor_Rodillos_pallets_vacios  ; Motor transporte de rodillos pallets vacios

